# EPICS substitutions: dpu3/Db/dpu3.substitutions
file "dpu3-det.template" { pattern
{P      DET     ADDR    VER}
{$(P)	$(DET1)	0	$(PROT_VER)}
{$(P)	$(DET2)	1	$(PROT_VER)}
{$(P)	$(DET3)	2	$(PROT_VER)}
{$(P)	$(DET4)	3	$(PROT_VER)}
}
